FUNCTION Event_add : BOOL
VAR_INPUT
	event	: ST_EVENT;
END_VAR
VAR
	i :INT;
END_VAR

//write event
FOR i:=0 TO GVL.iAlarm_max DO
	IF GVL.events_alarm[i].sEvent_MSG='' THEN
		GVL.events_alarm[i]	:= event;
		EXIT;
	END_IF
END_FOR
//check full
IF GVL.events_alarm[GVL.iAlarm_max].sEvent_MSG<>'' THEN
	FOR i:=0 TO GVL.iAlarm_max-1 DO
		GVL.events_alarm[i]	:= GVL.events_alarm[i+1];
	END_FOR
	GVL.events_alarm[GVL.iAlarm_max]	:= GVL.event_for_clear;
END_IF

END_FUNCTION

(* stored: Version 1.1.0.1, ProductVersion 3.1.4024.12
   POU Event_add: Id {bb8ccdbc-e3ad-4581-b2be-7d849efd6d91}, SpecialFunc None *)
